PROGRAM DewateringProcess
VAR
	fbRouteManager			:	FB_RouteManager;
	fbProcessDiagnostics	:	FB_ProcessDiagnostics;
	fbDeviceDiagnostics		:	FB_DeviceDiagnostics;
	fbMainProcessSupervisor	:	FB_MainProcessSupervisor;
	
	fbDischargeR01ToVR01	:	FB_DischargeR01ToVR01;
	
	fbBigBagDischarge		:	FB_BigBagDischarge;
	fbBigBagMassBalance			:   FB_BigBagMassBalance;  			
	

END_VAR

ACT_DeviceDiagnostics();
ACT_ProcessDiagnostics();
ACT_RouteManager();
ACT_MainProcessSupervisor();

ACT_BigBagDischarge();
ACT_BigBagMassBalance();

//ACT_BigBagFilling();

ACTION ACT_BigBagDischarge:
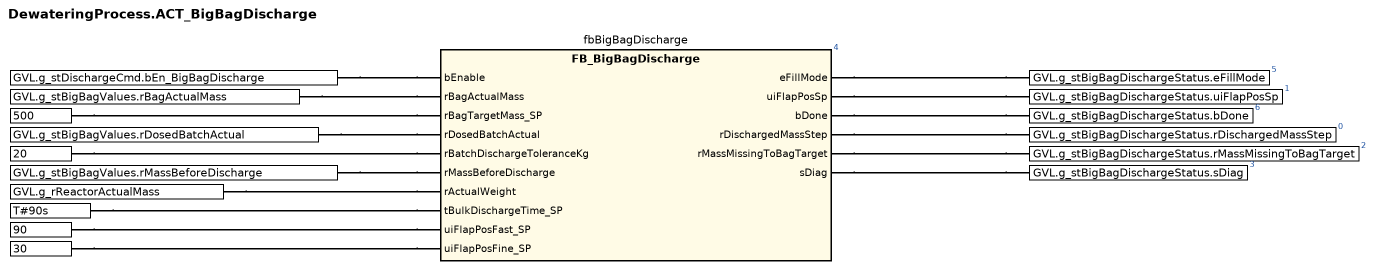
GVL.g_stBigBagDischargeStatus.rDischargedMassStep := fbBigBagDischarge.rDischargedMassStep;
GVL.g_stBigBagDischargeStatus.uiFlapPosSp := fbBigBagDischarge.uiFlapPosSp;
GVL.g_stBigBagDischargeStatus.rMassMissingToBagTarget := fbBigBagDischarge.rMassMissingToBagTarget;
GVL.g_stBigBagDischargeStatus.sDiag := fbBigBagDischarge.sDiag;
fbBigBagDischarge(
    bEnable := GVL.g_stDischargeCmd.bEn_BigBagDischarge,
    rBagActualMass := GVL.g_stBigBagValues.rBagActualMass,
    rBagTargetMass_SP := 500,
    rDosedBatchActual := GVL.g_stBigBagValues.rDosedBatchActual,
    rBatchDischargeToleranceKg := 20,
    rMassBeforeDischarge := GVL.g_stBigBagValues.rMassBeforeDischarge,
    rActualWeight := GVL.g_rReactorActualMass,
    tBulkDischargeTime_SP := T#90s,
    uiFlapPosFast_SP := 90,
    uiFlapPosFine_SP := 30); // FB_BigBagDischarge
GVL.g_stBigBagDischargeStatus.eFillMode := fbBigBagDischarge.eFillMode;
GVL.g_stBigBagDischargeStatus.bDone := fbBigBagDischarge.bDone;
END_ACTION

ACTION ACT_BigBagFilling:
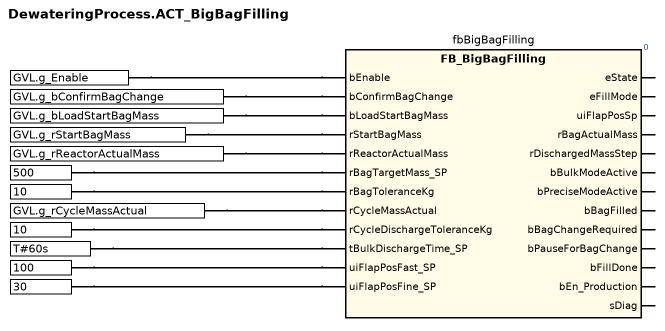
fbBigBagFilling(
    bEnable := GVL.g_Enable,
    bConfirmBagChange := GVL.g_bConfirmBagChange,
    bLoadStartBagMass := GVL.g_bLoadStartBagMass,
    rStartBagMass := GVL.g_rStartBagMass,
    rReactorActualMass := GVL.g_rReactorActualMass,
    rBagTargetMass_SP := 500,
    rBagToleranceKg := 10,
    rCycleMassActual := GVL.g_rCycleMassActual,
    rCycleDischargeToleranceKg := 10,
    tBulkDischargeTime_SP := T#60s,
    uiFlapPosFast_SP := 100,
    uiFlapPosFine_SP := 30); // FB_BigBagFilling
END_ACTION

ACTION ACT_BigBagMassBalance:
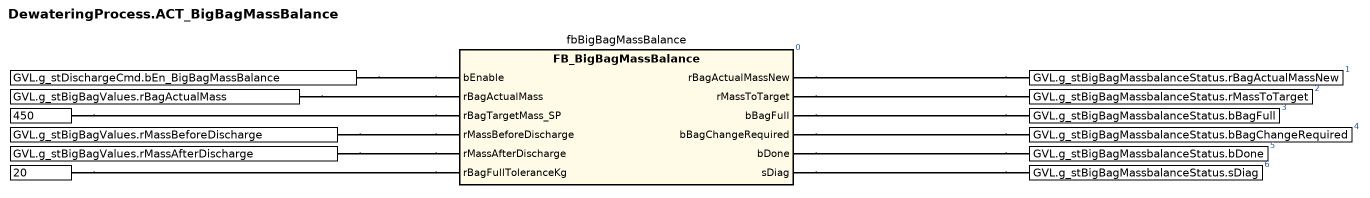
fbBigBagMassBalance(
    bEnable := GVL.g_stDischargeCmd.bEn_BigBagMassBalance,
    rBagActualMass := GVL.g_stBigBagValues.rBagActualMass,
    rBagTargetMass_SP := 450,
    rMassBeforeDischarge := GVL.g_stBigBagValues.rMassBeforeDischarge,
    rMassAfterDischarge := GVL.g_stBigBagValues.rMassAfterDischarge,
    rBagFullToleranceKg := 20); // FB_BigBagMassBalance
GVL.g_stBigBagMassbalanceStatus.rBagActualMassNew := fbBigBagMassBalance.rBagActualMassNew;
GVL.g_stBigBagMassbalanceStatus.rMassToTarget := fbBigBagMassBalance.rMassToTarget;
GVL.g_stBigBagMassbalanceStatus.bBagFull := fbBigBagMassBalance.bBagFull;
GVL.g_stBigBagMassbalanceStatus.bBagChangeRequired := fbBigBagMassBalance.bBagChangeRequired;
GVL.g_stBigBagMassbalanceStatus.bDone := fbBigBagMassBalance.bDone;
GVL.g_stBigBagMassbalanceStatus.sDiag := fbBigBagMassBalance.sDiag;
END_ACTION

ACTION ACT_DeviceDiagnostics:
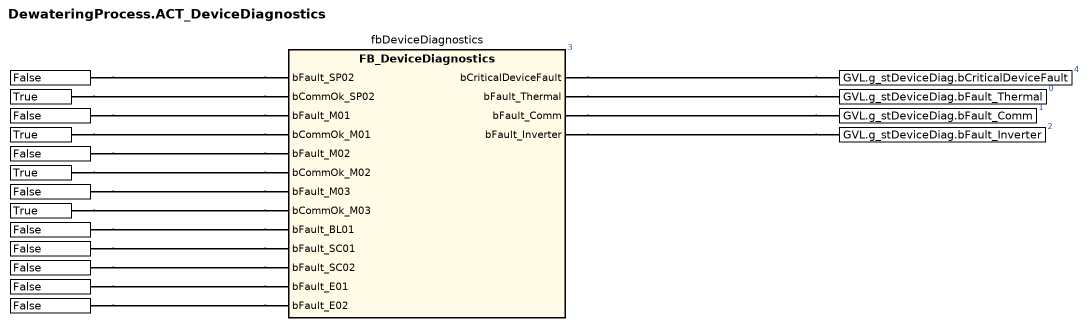
GVL.g_stDeviceDiag.bFault_Thermal := fbDeviceDiagnostics.bFault_Thermal;
GVL.g_stDeviceDiag.bFault_Comm := fbDeviceDiagnostics.bFault_Comm;
GVL.g_stDeviceDiag.bFault_Inverter := fbDeviceDiagnostics.bFault_Inverter;
fbDeviceDiagnostics(
    bFault_SP02 := False,
    bCommOk_SP02 := True,
    bFault_M01 := False,
    bCommOk_M01 := True,
    bFault_M02 := False,
    bCommOk_M02 := True,
    bFault_M03 := False,
    bCommOk_M03 := True,
    bFault_BL01 := False,
    bFault_SC01 := False,
    bFault_SC02 := False,
    bFault_E01 := False,
    bFault_E02 := False); // FB_DeviceDiagnostics
GVL.g_stDeviceDiag.bCriticalDeviceFault := fbDeviceDiagnostics.bCriticalDeviceFault;
END_ACTION

ACTION ACT_MainProcessSupervisor:
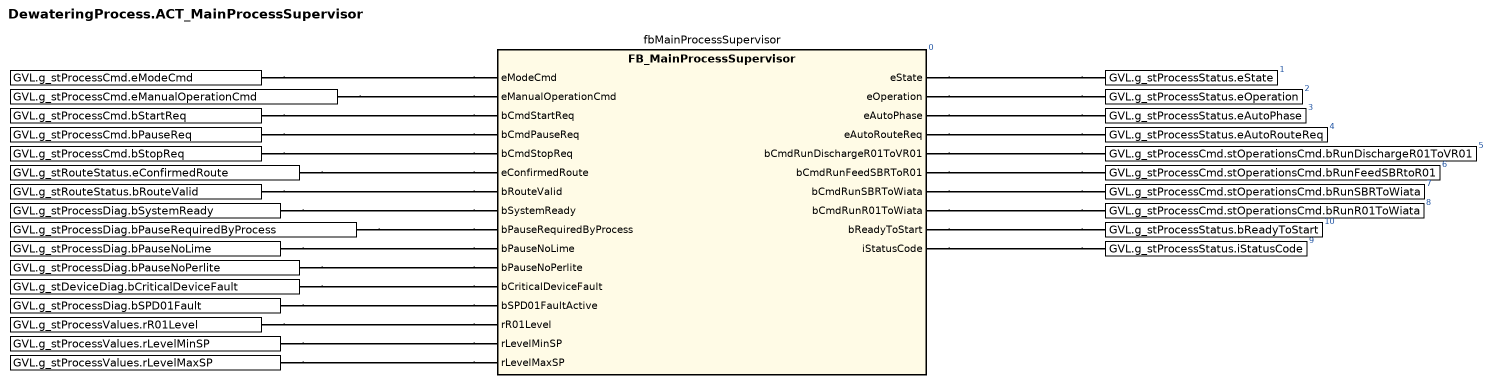
fbMainProcessSupervisor(
    eModeCmd := GVL.g_stProcessCmd.eModeCmd,
    eManualOperationCmd := GVL.g_stProcessCmd.eManualOperationCmd,
    bCmdStartReq := GVL.g_stProcessCmd.bStartReq,
    bCmdPauseReq := GVL.g_stProcessCmd.bPauseReq,
    bCmdStopReq := GVL.g_stProcessCmd.bStopReq,
    eConfirmedRoute := GVL.g_stRouteStatus.eConfirmedRoute,
    bRouteValid := GVL.g_stRouteStatus.bRouteValid,
    bSystemReady := GVL.g_stProcessDiag.bSystemReady,
    bPauseRequiredByProcess := GVL.g_stProcessDiag.bPauseRequiredByProcess,
    bPauseNoLime := GVL.g_stProcessDiag.bPauseNoLime,
    bPauseNoPerlite := GVL.g_stProcessDiag.bPauseNoPerlite,
    bCriticalDeviceFault := GVL.g_stDeviceDiag.bCriticalDeviceFault,
    bSPD01FaultActive := GVL.g_stProcessDiag.bSPD01Fault,
    rR01Level := GVL.g_stProcessValues.rR01Level,
    rLevelMinSP := GVL.g_stProcessValues.rLevelMinSP,
    rLevelMaxSP := GVL.g_stProcessValues.rLevelMaxSP); // FB_MainProcessSupervisor
GVL.g_stProcessStatus.eState := fbMainProcessSupervisor.eState;
GVL.g_stProcessStatus.eOperation := fbMainProcessSupervisor.eOperation;
GVL.g_stProcessStatus.eAutoPhase := fbMainProcessSupervisor.eAutoPhase;
GVL.g_stProcessStatus.eAutoRouteReq := fbMainProcessSupervisor.eAutoRouteReq;
GVL.g_stProcessCmd.stOperationsCmd.bRunDischargeR01ToVR01 := fbMainProcessSupervisor.bCmdRunDischargeR01ToVR01;
GVL.g_stProcessCmd.stOperationsCmd.bRunFeedSBRtoR01 := fbMainProcessSupervisor.bCmdRunFeedSBRToR01;
GVL.g_stProcessCmd.stOperationsCmd.bRunSBRToWiata := fbMainProcessSupervisor.bCmdRunSBRToWiata;
GVL.g_stProcessCmd.stOperationsCmd.bRunR01ToWiata := fbMainProcessSupervisor.bCmdRunR01ToWiata;
GVL.g_stProcessStatus.iStatusCode := fbMainProcessSupervisor.iStatusCode;
GVL.g_stProcessStatus.bReadyToStart := fbMainProcessSupervisor.bReadyToStart;
END_ACTION

ACTION ACT_ProcessDiagnostics:
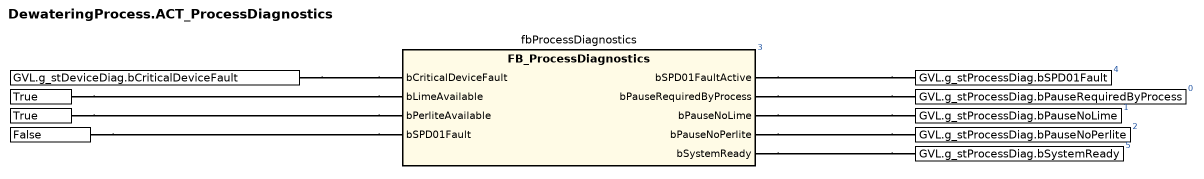
GVL.g_stProcessDiag.bPauseRequiredByProcess := fbProcessDiagnostics.bPauseRequiredByProcess;
GVL.g_stProcessDiag.bPauseNoLime := fbProcessDiagnostics.bPauseNoLime;
GVL.g_stProcessDiag.bPauseNoPerlite := fbProcessDiagnostics.bPauseNoPerlite;
fbProcessDiagnostics(
    bCriticalDeviceFault := GVL.g_stDeviceDiag.bCriticalDeviceFault,
    bLimeAvailable := True,
    bPerliteAvailable := True,
    bSPD01Fault := False); // FB_ProcessDiagnostics
GVL.g_stProcessDiag.bSPD01Fault := fbProcessDiagnostics.bSPD01FaultActive;
GVL.g_stProcessDiag.bSystemReady := fbProcessDiagnostics.bSystemReady;
END_ACTION

ACTION ACT_RouteManager:
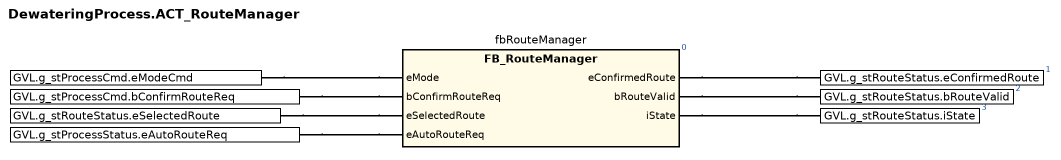
fbRouteManager(
    eMode := GVL.g_stProcessCmd.eModeCmd,
    bConfirmRouteReq := GVL.g_stProcessCmd.bConfirmRouteReq,
    eSelectedRoute := GVL.g_stRouteStatus.eSelectedRoute,
    eAutoRouteReq := GVL.g_stProcessStatus.eAutoRouteReq); // FB_RouteManager
GVL.g_stRouteStatus.eConfirmedRoute := fbRouteManager.eConfirmedRoute;
GVL.g_stRouteStatus.bRouteValid := fbRouteManager.bRouteValid;
GVL.g_stRouteStatus.iState := fbRouteManager.iState;
END_ACTION

END_PROGRAM

(* stored: Version 1.1.0.1, ProductVersion 3.1.4024.16
   POU DewateringProcess: Id {78b8de70-859f-4590-983a-34d148c9f601}, SpecialFunc None
   Action ACT_BigBagDischarge: Id {6da2ba3c-9242-4ae5-8ad1-27d6f7de8a96}
   Action ACT_BigBagFilling: Id {f8e8030a-066d-4a50-99e4-77b290311a8c}
   Action ACT_BigBagMassBalance: Id {9150b746-5e49-4d05-b69a-d3b0d3e0fa5c}
   Action ACT_DeviceDiagnostics: Id {7358511e-5737-4e7d-a07b-ad44094085d4}
   Action ACT_MainProcessSupervisor: Id {2f7e777b-8864-418d-b86d-a247dcca48c8}
   Action ACT_ProcessDiagnostics: Id {1103ca5c-4a87-4311-8acf-239e3bb2373f}
   Action ACT_RouteManager: Id {1a8a246c-4c55-4861-a582-2f60712a3f47} *)
